SYSTEM ExampleFbNetwork
  (* Version 1.0, 2022-05-12, AK115394 *)
  APPLICATION ExampleFbNetworkApp
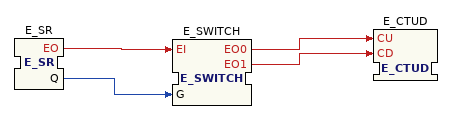
    FBS
      E_SR : E_SR;
      E_SWITCH : E_SWITCH;
      E_CTUD : E_CTUD;
    END_FBS
    EVENT_CONNECTIONS
      E_SR.EO TO E_SWITCH.EI;
      E_SWITCH.EO0 TO E_CTUD.CU;
      E_SWITCH.EO1 TO E_CTUD.CD;
    END_CONNECTIONS
    DATA_CONNECTIONS
      E_SR.Q TO E_SWITCH.G;
    END_CONNECTIONS
  END_APPLICATION
END_SYSTEM
